// TIA Portal V19 export
DATA_BLOCK "TestVersionControl_DB"   // DB2
// stored: InstanceOfName TestVersionControl, InstanceOfType FB
"TestVersionControl"
   // VAR_INPUT
   //    xStart : Bool;
   // END_VAR
   // VAR_OUTPUT
   //    xDiode : Bool;
   // END_VAR
BEGIN
END_DATA_BLOCK
